FUNCTION_BLOCK FbDelayN // Блок задержки сигнала на 100 тактов.

//      DbDelayN
//    +----------+
//    | FbDelayN |
// ->-|In     Out|->-
//    +----------+

VAR_INPUT //Входные переменные, сохраняемые.
In :REAL := 0.0; //Вход.
END_VAR

VAR_OUTPUT //Выходные переменные, сохраняемые.
Out :REAL := 0.0; //Выход.
END_VAR

CONST //Константы.
NUMBER := 98; //Размер массива Тактов 100 - 2 = 98.
END_CONST

VAR //Внутренние переменные, сохраняемые.
Buffer1: ARRAY [0..NUMBER] OF REAL; //Буфер задержки сигнала.
Counter1 :INT := 0; //Счетчик.
END_VAR

//W(Z)=Z^(-N), N=NUMBER+2
Out := Buffer1[NUMBER];
FOR COUNTER1 := NUMBER TO 1 BY -1 DO
Buffer1[COUNTER1] := Buffer1[Counter1 - 1];
END_FOR;
Buffer1[0] := In;

END_FUNCTION_BLOCK

//  +---------+
//  | GNU GPL |
//  +---------+
//  |
//  |
//  .= .-_-. =.
// ((_/)o o(\_))
//  `-'(. .)`-'
//  |/| \_/ |\
//  ( |     | )
//  /"\_____/"\
//  \__)   (__/
